(* IEC 61131-3 sources: nvidia-ai-factory-controls/libraries/AIFactory_Communication/POUs/DataEngine, 4 files *)

(* ---- GVL_PeerExchange.gvl ---- *)
(* =============================================================================
    GVL_PeerExchange — Inter-IPC Peer Data Exchange Buffer
    Common Library | NVIDIA AI Factory Controls
   =============================================================================

   PURPOSE:
     Shared memory for peer-to-peer IPC communication.
     Written by the Control_Task (fastest), read by all tasks.

   DATA FLOW:
     Control_Task writes stMyData → FB_PeerExchange sends to network
     FB_PeerExchange receives from network → writes astPeerData
     All tasks read astPeerData for their peer coordination needs

   TOPOLOGY:
     ┌─────────┐         UDP/OPC UA          ┌─────────┐
     │ IPC-01  │◄════════════════════════════►│ IPC-02  │
     │ (Power) │         Full Mesh            │(Cooling)│
     └────┬────┘                              └────┬────┘
          │           ┌─────────┐                  │
          └══════════►│ IPC-04  │◄═════════════════┘
                      │ (Safety)│
          ┌══════════►│         │◄═════════════════┐
          │           └────┬────┘                  │
     ┌────┴────┐           │                 ┌────┴────┐
     │ IPC-03  │◄══════════╝                 │  Edge   │
     │(Environ)│                             │ Gateway │
     └─────────┘                             └─────────┘

   SAFETY INVARIANT:
     If GVL_PeerExchange.bAllPeersSafetyOK = FALSE, the local IPC
     MUST enter degraded operation or safe-state (depending on subsystem).

   THREAD SAFETY:
     ST_PeerData is 128 bytes — fits in a cache line on most platforms.
     Written as atomic struct copy by owning task. Read by others at
     their cycle boundaries (cooperative scheduling ensures consistency).
   ============================================================================= *)

{attribute 'qualified_only'}
VAR_GLOBAL
    (* ─── My Outbound Data (populated by Control_Task) ─── *)
    stMyData             : ST_PeerData;

    (* ─── Received Peer Data (populated by PeerExchange FB) ─── *)
    stPeer_Power         : ST_PeerData;     (* From IPC-01 *)
    stPeer_Cooling       : ST_PeerData;     (* From IPC-02 *)
    stPeer_Environment   : ST_PeerData;     (* From IPC-03 *)
    stPeer_Safety        : ST_PeerData;     (* From IPC-04 *)

    (* ─── Aggregate Status (computed by PeerExchange FB) ─── *)
    bAllPeersSafetyOK    : BOOL := TRUE;    (* All peers permit operation *)
    bAnyPeerEmergency    : BOOL := FALSE;   (* Any peer in emergency *)
    bAnyPeerDead         : BOOL := FALSE;   (* Any peer not responding *)

    (* ─── Per-Peer Health ─── *)
    bPeer_Power_Alive    : BOOL;
    bPeer_Cooling_Alive  : BOOL;
    bPeer_Environment_Alive : BOOL;
    bPeer_Safety_Alive   : BOOL;

    (* ─── Cross-IPC Coordination Commands ─── *)
    (* These are SET by one IPC and READ by another for real-time coordination *)
    bCmd_PowerShed       : BOOL;            (* Cooling→Power: need load reduction *)
    bCmd_MaxCool         : BOOL;            (* Power→Cooling: thermal emergency *)
    bCmd_StopCooling     : BOOL;            (* Safety→Cooling: stop pumps (leak) *)
    bCmd_EmergencyVent   : BOOL;            (* Safety→Environment: start purge fans *)
END_VAR

(* ---- FB_DataCollector.fb ---- *)
(* =============================================================================
    FB_DataCollector — Multi-Protocol Data Collection & Publishing Engine
    Common Library | NVIDIA AI Factory Controls
   =============================================================================

   PURPOSE:
     Central data broker that:
       1. COLLECTS data from control FBs (via GVL_CrossTask snapshots)
       2. EVALUATES publish conditions (deadband, timing, change-of-value)
       3. DISPATCHES to multiple publishers simultaneously (fan-out)
       4. RECEIVES data from external sources via subscribers (fan-in)

   ARCHITECTURE:
     ┌──────────────────────────────────────────────────────────────────┐
     │                    FB_DataCollector                               │
     │                                                                  │
     │  ┌─────────────┐    ┌──────────────┐    ┌──────────────────┐   │
     │  │ Data Points │    │  Publish     │    │  Publishers[]    │   │
     │  │ Registry    │───→│  Engine      │───→│  (I_DataPublisher)│   │
     │  │ (ST_Data    │    │  (deadband,  │    │  ├─ OPC UA       │   │
     │  │  Point[])   │    │   timing,    │    │  ├─ MQTT         │   │
     │  │             │    │   CoV eval)  │    │  ├─ Modbus       │   │
     │  └─────────────┘    └──────────────┘    │  └─ SharedMem    │   │
     │                                          └──────────────────┘   │
     │  ┌─────────────────────────────────────────────────────────┐   │
     │  │  Subscribers[] (I_DataSubscriber)                        │   │
     │  │  ├─ OPC UA client (other IPCs)                          │   │
     │  │  ├─ MQTT subscribe (cloud commands)                     │   │
     │  │  └─ REST client (GPU telemetry)                         │   │
     │  └─────────────────────────────────────────────────────────┘   │
     └──────────────────────────────────────────────────────────────────┘

   MULTI-PROTOCOL CHOICE:
     Publishers and subscribers are registered at startup via
     M_AddPublisher / M_AddSubscriber. You can register ANY combination:
       • OPC UA only (traditional SCADA)
       • MQTT only (cloud-native)
       • OPC UA + MQTT (dual-path redundancy)
       • All protocols (maximum integration)

   PUBLISH MODES:
     CYCLIC     — Every N milliseconds, regardless of value change
     ON_CHANGE  — Only when value differs from last publish by > deadband
     HYBRID     — On-change with guaranteed heartbeat (max silence interval)
     ON_DEMAND  — Only when explicitly triggered (events, alarms)

   PERFORMANCE:
     At 100ms cycle with 500 data points:
       CYCLIC mode:    500 publishes/cycle = 5000/s (high bandwidth)
       ON_CHANGE mode: ~50 publishes/cycle = 500/s (typical)
       HYBRID mode:    ~80 publishes/cycle = 800/s (balanced)

   RACE CONDITION PREVENTION:
     • Runs in Communication_Task (100ms cycle, priority 5)
     • Reads from GVL_CrossTask at START of cycle (atomic struct copy)
     • Writes to GVL_CrossTask at END of cycle (subscriber data)
     • Never accesses control FB internals directly

   TASK ASSIGNMENT:
     Communication_Task — Priority 5, Cycle 100ms
   ============================================================================= *)

(* ═══════════════════════════════════════════════════════════════════════════════
   DECLARATION
   ═══════════════════════════════════════════════════════════════════════════════ *)

{attribute 'no_assign'}
FUNCTION_BLOCK FB_DataCollector EXTENDS FB_Base
VAR_INPUT
    (* --- Timing --- *)
    fCycleTime_s         : REAL := 0.1;     (* Communication task cycle [seconds] *)
    nSystemTime_ms       : UDINT;           (* System millisecond counter *)
END_VAR

VAR_OUTPUT
    (* --- Statistics --- *)
    nTotalPoints         : UINT;            (* Registered data points *)
    nPublishedThisCycle  : UINT;            (* Points published this scan *)
    nPublishErrors       : UDINT;           (* Cumulative publish failures *)
    nSubscribedPoints    : UINT;            (* Active subscriptions *)
    nStaleSubscriptions  : UINT;            (* Subscriptions with stale data *)
    nActivePublishers    : USINT;           (* Connected publishers *)
    nActiveSubscribers   : USINT;           (* Connected subscribers *)
END_VAR

VAR
    (* --- Data Point Registry --- *)
    _astPoints           : ARRAY[1..500] OF ST_DataPoint;  (* Max 500 points *)
    _nPointCount         : UINT;

    (* --- Publisher Registry (Strategy Pattern) --- *)
    _arefPublishers      : ARRAY[1..8] OF I_DataPublisher; (* Max 8 backends *)
    _nPublisherCount     : USINT;

    (* --- Subscriber Registry --- *)
    _arefSubscribers     : ARRAY[1..8] OF I_DataSubscriber; (* Max 8 sources *)
    _nSubscriberCount    : USINT;

    (* --- Internal --- *)
    _nPublishIndex       : UINT;            (* Current point being evaluated *)
    _nMaxPublishPerCycle : UINT := 100;     (* Throttle: max publishes per scan *)
    _nCyclePublishCount  : UINT;            (* Counter for this cycle *)
    _bBatchActive        : BOOL;            (* Batch mode active *)

    (* --- Loop Variables --- *)
    _i                   : UINT;
    _j                   : USINT;
END_VAR

VAR CONSTANT
    C_MAX_POINTS         : UINT := 500;
    C_MAX_PUBLISHERS     : USINT := 8;
    C_MAX_SUBSCRIBERS    : USINT := 8;
    C_QUALITY_GOOD       : USINT := 0;
    C_QUALITY_UNCERTAIN  : USINT := 1;
    C_QUALITY_BAD        : USINT := 2;
END_VAR

(* ═══════════════════════════════════════════════════════════════════════════════
   IMPLEMENTATION
   ═══════════════════════════════════════════════════════════════════════════════ *)

(* Lifecycle managed by FB_Base *)
SUPER^();

(* ---- FB_PeerExchange_OPCUA.fb ---- *)
(* =============================================================================
    FB_PeerExchange_OPCUA — OPC UA Direct Peer-to-Peer Exchange
    Common Library | NVIDIA AI Factory Controls
   =============================================================================

   PURPOSE:
     Implements I_PeerExchange using OPC UA client/server.
     Each IPC runs an OPC UA server exposing its ST_PeerData.
     Each IPC runs OPC UA clients reading peers' ST_PeerData.

   HOW IT WORKS:
     SEND: Write local ST_PeerData to GVL_PeerExchange.stMyData
           (OPC UA server exposes this variable automatically)

     RECEIVE: OPC UA client reads peer's stMyData variable every cycle.
              Result stored in GVL_PeerExchange.stPeer[n]_Data.

   LATENCY:
     OPC UA subscription at 5ms publishing interval → ~5-10ms latency.
     Acceptable for safety permit (< 10ms requirement).
     For sub-millisecond: use FB_PeerExchange_UDP instead.

   FAILOVER:
     If peer OPC UA server unreachable for > nTimeout_ms:
       • Mark peer as DEAD
       • Safety data: assume worst case (permit = FALSE)
       • Operational data: use last-known-good with STALE quality

   TOPOLOGY:
     IPC-01 ←──OPC UA──→ IPC-02
       ↕                    ↕
     IPC-04 ←──OPC UA──→ IPC-03

     Full mesh: each IPC connects to all other 3.
     N*(N-1) = 4*3 = 12 OPC UA client connections total.
   ============================================================================= *)

(* ═══════════════════════════════════════════════════════════════════════════════
   DECLARATION
   ═══════════════════════════════════════════════════════════════════════════════ *)

{attribute 'no_assign'}
FUNCTION_BLOCK FB_PeerExchange_OPCUA EXTENDS FB_Base IMPLEMENTS I_PeerExchange
VAR_INPUT
    (* --- Local IPC Identity --- *)
    nMyIPC_ID            : USINT := 2;      (* This IPC's ID (1-4) *)

    (* --- Peer Configuration --- *)
    asPeerURLs           : ARRAY[1..4] OF STRING(128);  (* OPC UA URLs *)
    asPeerNames          : ARRAY[1..4] OF STRING(32);   (* Logical names *)

    (* --- Timing --- *)
    fCycleTime_s         : REAL := 0.005;   (* Control task cycle *)
    nTimeout_ms          : UDINT := 50;     (* Peer timeout [ms] *)
    nSubscriptionRate_ms : UDINT := 5;      (* OPC UA subscription interval *)
END_VAR

VAR_OUTPUT
    (* --- Received Peer Data (one per peer IPC) --- *)
    astPeerData          : ARRAY[1..4] OF ST_PeerData;
    abPeerAlive          : ARRAY[1..4] OF BOOL;
    anPeerLatency_us     : ARRAY[1..4] OF UDINT;

    (* --- Aggregate Safety (pessimistic across all peers) --- *)
    bAllPeersSafetyOK    : BOOL;            (* TRUE only if ALL peers permit *)
    bAnyPeerEmergency    : BOOL;            (* TRUE if ANY peer has emergency *)
    bAnyPeerDead         : BOOL;            (* TRUE if ANY peer not responding *)

    (* --- My Published Data (what this IPC sends to peers) --- *)
    stMyData             : ST_PeerData;
END_VAR

VAR
    (* --- Per-Peer Connection State --- *)
    _abConnected         : ARRAY[1..4] OF BOOL;
    _anTimeSinceUpdate   : ARRAY[1..4] OF UDINT;  (* ms since last receive *)
    _anLastSequence      : ARRAY[1..4] OF UDINT;  (* Last received sequence # *)
    _anMissedPackets     : ARRAY[1..4] OF UDINT;  (* Gap in sequence counter *)

    (* --- Edge Triggers --- *)
    _artrigPeerLost      : ARRAY[1..4] OF R_TRIG; (* Peer went offline *)
    _artrigPeerFound     : ARRAY[1..4] OF R_TRIG; (* Peer came back online *)
    _rtrigEmergency      : R_TRIG;                (* Any peer raised emergency *)

    (* --- Sequence Counter --- *)
    _nMySequence         : UDINT;

    (* --- Loop Variable --- *)
    _i                   : USINT;
END_VAR

(* ═══════════════════════════════════════════════════════════════════════════════
   IMPLEMENTATION
   ═══════════════════════════════════════════════════════════════════════════════ *)

SUPER^();

(* ---- FB_PeerExchange_UDP.fb ---- *)
(* =============================================================================
    FB_PeerExchange_UDP — UDP Multicast Fast Peer Exchange
    Common Library | NVIDIA AI Factory Controls
   =============================================================================

   PURPOSE:
     Implements I_PeerExchange using raw UDP multicast for minimum latency.
     All IPCs join the same multicast group. Each broadcasts its ST_PeerData
     every control cycle. All peers receive simultaneously.

   LATENCY:
     UDP multicast on switched Ethernet: < 1ms (typically 100-500µs).
     This is 10-50x faster than OPC UA subscriptions.

   WHEN TO USE:
     • Safety permit propagation (hardwired is primary, UDP is backup)
     • Real-time load coordination between power and cooling
     • Sub-5ms response requirements

   WHEN NOT TO USE:
     • Across network segments (multicast doesn't cross routers by default)
     • When encryption is required (UDP multicast is unencrypted)
     • For large data payloads (keep to ST_PeerData size ~128 bytes)

   MULTICAST SETUP:
     Group: 239.192.100.1 (link-local multicast, stays on control VLAN)
     Port: 50100
     All IPCs join this group on their control network interface.

   PACKET FORMAT:
     [4 bytes: magic 0xAF5C] [2 bytes: length] [ST_PeerData] [2 bytes: CRC16]

   FAIL-SAFE:
     If no packet received from a peer within nTimeout_ms → peer is DEAD.
     Dead peer assumed to have revoked safety permit (pessimistic).

   REQUIRES:
     CODESYS SysSocket library for raw UDP socket operations.

   REDUNDANCY:
     Run BOTH FB_PeerExchange_OPCUA and FB_PeerExchange_UDP.
     Control logic uses the FRESHEST data from either source.
     If UDP fails: fall back to OPC UA (higher latency but still works).
     If OPC UA fails: fall back to UDP.
     If BOTH fail: hardwired safety signals are the last line of defense.
   ============================================================================= *)

(* ═══════════════════════════════════════════════════════════════════════════════
   DECLARATION
   ═══════════════════════════════════════════════════════════════════════════════ *)

{attribute 'no_assign'}
FUNCTION_BLOCK FB_PeerExchange_UDP EXTENDS FB_Base IMPLEMENTS I_PeerExchange
VAR_INPUT
    (* --- Network Configuration --- *)
    sMulticastGroup      : STRING(16) := '239.192.100.1';
    nPort                : UINT := 50100;
    sLocalInterface      : STRING(16) := '192.168.100.0';  (* Bind to control NIC *)

    (* --- Identity --- *)
    nMyIPC_ID            : USINT := 2;

    (* --- Timing --- *)
    fCycleTime_s         : REAL := 0.005;
    nTimeout_ms          : UDINT := 20;     (* 20ms = 4 missed packets at 5ms *)
END_VAR

VAR_OUTPUT
    (* --- Received Peer Data --- *)
    astPeerData          : ARRAY[1..4] OF ST_PeerData;
    abPeerAlive          : ARRAY[1..4] OF BOOL;
    anPeerLatency_us     : ARRAY[1..4] OF UDINT;

    (* --- Aggregate Safety --- *)
    bAllPeersSafetyOK    : BOOL;
    bAnyPeerEmergency    : BOOL;
    bAnyPeerDead         : BOOL;

    (* --- My Published Data --- *)
    stMyData             : ST_PeerData;

    (* --- Network Stats --- *)
    nPacketsSent         : UDINT;
    nPacketsReceived     : UDINT;
    nPacketsDropped      : UDINT;           (* CRC errors or invalid *)
    nSequenceGaps        : UDINT;           (* Missed packets total *)
END_VAR

VAR
    (* --- Socket Handle --- *)
    _hSocket             : UDINT;           (* SysSocket handle *)
    _bSocketOpen         : BOOL;

    (* --- Per-Peer Tracking --- *)
    _anTimeSinceUpdate   : ARRAY[1..4] OF UDINT;
    _anLastSequence      : ARRAY[1..4] OF UDINT;

    (* --- Transmit Buffer --- *)
    _abTxBuffer          : ARRAY[0..255] OF BYTE;
    _nTxSize             : UINT;

    (* --- Receive Buffer --- *)
    _abRxBuffer          : ARRAY[0..255] OF BYTE;
    _nRxSize             : UINT;

    (* --- Sequence --- *)
    _nMySequence         : UDINT;

    (* --- Edge Triggers --- *)
    _artrigPeerLost      : ARRAY[1..4] OF R_TRIG;
    _rtrigEmergency      : R_TRIG;

    (* --- CRC --- *)
    _nCRC                : WORD;

    (* --- Loop --- *)
    _i                   : USINT;
END_VAR

VAR CONSTANT
    C_MAGIC              : DWORD := 16#AF5C0000;  (* Packet magic number *)
    C_MAX_PACKET         : UINT := 200;            (* Max packet size *)
END_VAR

(* ═══════════════════════════════════════════════════════════════════════════════
   IMPLEMENTATION
   ═══════════════════════════════════════════════════════════════════════════════ *)

(* In production with CODESYS SysSocket library:

   1. M_Initialize:
      - Open UDP socket
      - Join multicast group
      - Set socket to non-blocking

   2. M_Execute (every 5ms cycle):
      a) SEND: serialize stMyData → _abTxBuffer, append CRC, sendto multicast
      b) RECEIVE: recvfrom (non-blocking), parse, validate CRC, update astPeerData
      c) TIMEOUT: check per-peer freshness, mark dead if stale
      d) SAFETY: compute aggregate safety state (same logic as OPCUA version)

   3. M_SafeState:
      - Close socket
      - Mark all peers dead
      - Assume worst-case safety
*)

SUPER^();
